Fanuc KAREL source: kt00058.KL

-- PROVISIONAL review KL for V1013-1; original PC SHA256 b19771ccbc138bfbb1038a7aa60964767d6dd9a9c81289518f9e51da3fbc5cac
-- Incomplete behavior may be omitted. Consult companion uncertainty JSON. Do not deploy.
PROGRAM KT00058
%NOLOCKGROUP
VAR
  I2 : INTEGER
  OUT : REAL
-- UNRESOLVED_DECL H1 type=002017
BEGIN
  -- UNRESOLVED_PC offsets 5-19; opcodes 2E,22,9D,33,B4
  -- UNRESOLVED_PC offsets 24-35; opcodes 2E,23
  -- UNRESOLVED_PC offsets 40-63; opcodes 22,9D,33,B3,21,53,64,23
  -- UNRESOLVED_PC offsets 68-72; opcodes 7F
END KT00058
